{attribute addProperty BoxType "EL6224-0090-0016"}
{attribute addProperty Id "Module_1_DeviceState_Inputs_DeviceModule_1_DeviceState_Inputs_Device_50DD3C951620Module_2_DeviceState_InputsModule_2_DeviceState_Inputs_D860B2E33240WcStateAT %I*WcState_F855686C1620InfoDataAT %I*InfoData_275E3363128160"}
{attribute addProperty CRC "3745819289"}
{attribute addProperty SizeInBites "192"}
{attribute addProperty SizeInBytes "24"}
TYPE EL6224_193A1401 :
STRUCT
	{attribute addProperty Name "Module_1_DeviceState_Inputs_Device"}
	Module_1_DeviceState_Inputs_Device : Module_1_DeviceState_Inputs_Device_50DD3C95;
	{attribute addProperty Name "Module_2_DeviceState_Inputs"}
	Module_2_DeviceState_Inputs : Module_2_DeviceState_Inputs_D860B2E3;
	{attribute addProperty Name "WcState"}
	WcState : WcState_F855686C;
	{attribute addProperty Name "InfoData"}
	InfoData : InfoData_275E3363;
END_STRUCT
END_TYPE

(* stored: Version 1.2.0.0, ProductVersion 3.1.4024.9
   DUT EL6224_193A1401: Id {09967919-d5ac-4619-81c1-0cfecda24acc} *)
